// TIA Portal V20 export
// export: Created 2026-05-08T20:35:38.5773715Z, ExportSetting WithDefaults, DisplayName Totally Integrated Automation Portal, DisplayVersion V20 Update 4, DisplayName TIA Portal Openness, DisplayVersion V20 Update 4, DisplayName TIA Portal Version Control Interface, DisplayVersion V20 Update 4, DisplayName SINAMICS Startdrive Advanced, DisplayVersion V20 SP1 Update 2, DisplayName SINAMICS Startdrive G110M, G120, G120C, G120D, G120P, G115D, DisplayVersion V20 SP1 Update 2, DisplayName SINAMICS Startdrive G130, G150, S120, S150, SINAMICS MV, G220, S200, S210, DisplayVersion V20 SP1 Update 2, DisplayName STEP 7 Professional, DisplayVersion V20 Update 4, DisplayName STEP 7 Safety, DisplayVersion V20 Update 2, DisplayName WinCC Basic/Comfort/Advanced, DisplayVersion V20 Update 4, DisplayName SIMATIC Visualization Architect, DisplayVersion V20 Update 4, DisplayName WinCC Unified, DisplayVersion V20 Update 4, DisplayName SIMATIC Visualization Architect, DisplayVersion V20 Update 4
TYPE "LDrive_typeKistlerHmi"
// stored: IsFailsafeCompliant false
   STRUCT
      state : DWord;   // State tec_unit
      plantidentifier : WString[24];
      move : Word;   // Interface Movement Position
      alarm : DWord;
      stateColour : SInt;
      receive : Struct
         status : DWord;
         mpNum : Byte;
         cfgMpNum : Byte;
         cfgAddress : Byte;
         cfgLength : Byte;
         selectPage : Byte;
         selectSequence : Byte;
         PVcurrentValueX : Real;
         PVcurrentValueY : Real;
         "PVcurrentXmin-X" : Real;
         "PVcurrentXmax-X" : Real;
         "PVcurrentYmin-Y" : Real;
         "PVcurrentYmax-Y" : Real;
         serverJogSpeed : Real;   // mm/s
         serverJogMaxForce : Real;
         PV_EO1_Force { ExternalVisible := 'False'; ExternalWritable := 'False'} : Real;
         PV_EO2_Distance { ExternalVisible := 'False'; ExternalWritable := 'False'} : Real;
         PV_EO3_Gradient { ExternalVisible := 'False'; ExternalWritable := 'False'} : Real;
         PV_Real_EO7 { ExternalVisible := 'False'; ExternalWritable := 'False'} : Real;
         PV_Real_EO8 { ExternalVisible := 'False'; ExternalWritable := 'False'} : Real;
         PV_Real_EO9 { ExternalVisible := 'False'; ExternalWritable := 'False'} : Real;
         PV_Real_E10 { ExternalVisible := 'False'; ExternalWritable := 'False'} : Real;
         PV_E04_Nopass { ExternalVisible := 'False'; ExternalWritable := 'False'} : Byte;
         PV_E05_Unibox { ExternalVisible := 'False'; ExternalWritable := 'False'} : Byte;
         PV_E06_Envelope { ExternalVisible := 'False'; ExternalWritable := 'False'} : Byte;
         PV_Byte_E07 { ExternalVisible := 'False'; ExternalWritable := 'False'} : Byte;
         PV_Byte_E08 { ExternalVisible := 'False'; ExternalWritable := 'False'} : Byte;
         PV_Byte_E09 { ExternalVisible := 'False'; ExternalWritable := 'False'} : Byte;
         PV_Byte_E10 { ExternalVisible := 'False'; ExternalWritable := 'False'} : Byte;
      END_STRUCT;
      send : Struct
         control : DWord;
         mpNum : Byte;
         cfgMpNum : Byte;
         cfgAddress : Byte;
         cfgLength : Byte;
         selectPage : Byte;
         selectSeqeunce : Byte;
         serverJogSpeed : Real;
         serverJogMaxForce : Real;
      END_STRUCT;
      serverJogSpeedSet : Real;
      serverJogMaxForceSet : Real;
      cfgMpNumSet : Byte;
      cfgAddressSet : Byte;
      cfgLengthSet : Byte;
      selectPageSet : Byte;
      selectSequenceSet : Byte;
      manualSelectMpNum : Byte;
      currentLabel : Byte;
      sequenceEnd : Bool;
      hmiControlNo : Int;
      opmodearea : USInt;
      select : Bool;
      hmiSelectWord : Word;
      tecUnitNumber : Int;
      codeViewCondControl : Struct
         advanceConditions : Bool;
         reverseConditions : Bool;
         condiitonsFilter : WString[48];
      END_STRUCT;
      ipAddressplant : String;
   END_STRUCT;
END_TYPE
